(* IEC 61131-3 sources: 2026_Projet_YGO_ExcavatriceDragage/TOOLS/TEST_AUTO_CI/RESULTS/JOYSTICK/tests, 1 file *)

(* ---- test_fb_joystick.st ---- *)
SETUP
VAR
    fb : FB_JOYSTICK;
    nx : INT := 5000;
    ny : INT := 5000;
    diagOk : ST_DIAG_DEVICE;
    diagDown : ST_DIAG_DEVICE;
END_VAR
END_SETUP

TEST 'TC-P08-001 Bus non operationnel neutralise les sorties sans lever Error'
    diagDown.ONLINE := FALSE; diagDown.OPERATIONAL := FALSE; diagDown.ERROR := FALSE;
    diagDown.ERRORID := 0; diagDown.STATE := E_DIAG_STATE.INIT; diagDown.STATEATERROR := E_DIAG_STATE.DISABLED;
    diagOk.ONLINE := TRUE; diagOk.OPERATIONAL := TRUE; diagOk.ERROR := FALSE;
    diagOk.ERRORID := 0; diagOk.STATE := E_DIAG_STATE.READY; diagOk.STATEATERROR := E_DIAG_STATE.DISABLED;

    fb(ENABLE := TRUE, RESET := FALSE, POWERCONTACTORENGAGED := TRUE,
       MODE := E_MODE.MAINT_N1, BENNEBUSY := FALSE, PRESERVEARMINGAFTERBUCKET := FALSE,
       BUSCANOPENOP := diagDown, JOYSTICKOP := diagOk,
       RAWX := 5000, RAWY := 5000, RAWBUTTON := FALSE, BTNCALIBRATE := FALSE,
       INVERTX := FALSE, INVERTY := FALSE, DEADBANDRAW := 300, FILTERTIME := T#0MS,
       NEUTRALHOLDTIME := T#100MS, DEADMANARMHOLDTIME := T#100MS, DEADMANARMGRACETIME := T#3S,
       NEUTRALXMEM := nx, NEUTRALYMEM := ny);

    ASSERT_FALSE(fb.READY, 'bus CAN non operationnel doit bloquer Ready');
    ASSERT_FALSE(fb.ERROR, 'un bus down est un GATE de securite, PAS une Error diagnostiquee (pas de bit ErrorId leve ici)');
    ASSERT_FALSE(fb.AXISCMDX.ENABLE, 'sorties axe neutralisees si non operationnel');
END_TEST

TEST 'TC-P08-002 Appui maintenu 100ms arme le geste (DeadmanArmHoldTime)'
    diagOk.ONLINE := TRUE; diagOk.OPERATIONAL := TRUE; diagOk.ERROR := FALSE;
    diagOk.ERRORID := 0; diagOk.STATE := E_DIAG_STATE.READY; diagOk.STATEATERROR := E_DIAG_STATE.DISABLED;

    (* baseline : neutre, bouton relache *)
    fb(ENABLE := TRUE, RESET := FALSE, POWERCONTACTORENGAGED := TRUE,
       MODE := E_MODE.MAINT_N1, BENNEBUSY := FALSE, PRESERVEARMINGAFTERBUCKET := FALSE,
       BUSCANOPENOP := diagOk, JOYSTICKOP := diagOk,
       RAWX := 5000, RAWY := 5000, RAWBUTTON := FALSE, BTNCALIBRATE := FALSE,
       INVERTX := FALSE, INVERTY := FALSE, DEADBANDRAW := 300, FILTERTIME := T#0MS,
       NEUTRALHOLDTIME := T#100MS, DEADMANARMHOLDTIME := T#100MS, DEADMANARMGRACETIME := T#3S,
       NEUTRALXMEM := nx, NEUTRALYMEM := ny);
    ASSERT_FALSE(fb.DEADMANARMED, 'baseline : bouton relache, pas arme');

    (* front bouton : demarre le maintien, pas encore arme *)
    fb(ENABLE := TRUE, RESET := FALSE, POWERCONTACTORENGAGED := TRUE,
       MODE := E_MODE.MAINT_N1, BENNEBUSY := FALSE, PRESERVEARMINGAFTERBUCKET := FALSE,
       BUSCANOPENOP := diagOk, JOYSTICKOP := diagOk,
       RAWX := 5000, RAWY := 5000, RAWBUTTON := TRUE, BTNCALIBRATE := FALSE,
       INVERTX := FALSE, INVERTY := FALSE, DEADBANDRAW := 300, FILTERTIME := T#0MS,
       NEUTRALHOLDTIME := T#100MS, DEADMANARMHOLDTIME := T#100MS, DEADMANARMGRACETIME := T#3S,
       NEUTRALXMEM := nx, NEUTRALYMEM := ny);
    ASSERT_FALSE(fb.DEADMANARMED, 'front bouton seul ne doit pas armer immediatement (maintien requis)');

    (* 50ms plus tard : maintien pas termine *)
    ADVANCE_TIME(50000000);
    fb(ENABLE := TRUE, RESET := FALSE, POWERCONTACTORENGAGED := TRUE,
       MODE := E_MODE.MAINT_N1, BENNEBUSY := FALSE, PRESERVEARMINGAFTERBUCKET := FALSE,
       BUSCANOPENOP := diagOk, JOYSTICKOP := diagOk,
       RAWX := 5000, RAWY := 5000, RAWBUTTON := TRUE, BTNCALIBRATE := FALSE,
       INVERTX := FALSE, INVERTY := FALSE, DEADBANDRAW := 300, FILTERTIME := T#0MS,
       NEUTRALHOLDTIME := T#100MS, DEADMANARMHOLDTIME := T#100MS, DEADMANARMGRACETIME := T#3S,
       NEUTRALXMEM := nx, NEUTRALYMEM := ny);
    ASSERT_FALSE(fb.DEADMANARMED, '50ms < DeadmanArmHoldTime (100ms) : pas encore arme');

    (* 60ms de plus (total 110ms) : maintien termine -> arme *)
    ADVANCE_TIME(60000000);
    fb(ENABLE := TRUE, RESET := FALSE, POWERCONTACTORENGAGED := TRUE,
       MODE := E_MODE.MAINT_N1, BENNEBUSY := FALSE, PRESERVEARMINGAFTERBUCKET := FALSE,
       BUSCANOPENOP := diagOk, JOYSTICKOP := diagOk,
       RAWX := 5000, RAWY := 5000, RAWBUTTON := TRUE, BTNCALIBRATE := FALSE,
       INVERTX := FALSE, INVERTY := FALSE, DEADBANDRAW := 300, FILTERTIME := T#0MS,
       NEUTRALHOLDTIME := T#100MS, DEADMANARMHOLDTIME := T#100MS, DEADMANARMGRACETIME := T#3S,
       NEUTRALXMEM := nx, NEUTRALYMEM := ny);
    ASSERT_TRUE(fb.DEADMANARMED, '110ms >= DeadmanArmHoldTime (100ms) : geste arme');
END_TEST

TEST 'TC-P08-003 Relachement du bouton avant fin du maintien annule la tentative armement'
    diagOk.ONLINE := TRUE; diagOk.OPERATIONAL := TRUE; diagOk.ERROR := FALSE;
    diagOk.ERRORID := 0; diagOk.STATE := E_DIAG_STATE.READY; diagOk.STATEATERROR := E_DIAG_STATE.DISABLED;

    (* front bouton : demarre le maintien *)
    fb(ENABLE := TRUE, RESET := FALSE, POWERCONTACTORENGAGED := TRUE,
       MODE := E_MODE.MAINT_N1, BENNEBUSY := FALSE, PRESERVEARMINGAFTERBUCKET := FALSE,
       BUSCANOPENOP := diagOk, JOYSTICKOP := diagOk,
       RAWX := 5000, RAWY := 5000, RAWBUTTON := TRUE, BTNCALIBRATE := FALSE,
       INVERTX := FALSE, INVERTY := FALSE, DEADBANDRAW := 300, FILTERTIME := T#0MS,
       NEUTRALHOLDTIME := T#100MS, DEADMANARMHOLDTIME := T#100MS, DEADMANARMGRACETIME := T#3S,
       NEUTRALXMEM := nx, NEUTRALYMEM := ny);

    (* relache a 50ms, avant la fin des 100ms de maintien *)
    ADVANCE_TIME(50000000);
    fb(ENABLE := TRUE, RESET := FALSE, POWERCONTACTORENGAGED := TRUE,
       MODE := E_MODE.MAINT_N1, BENNEBUSY := FALSE, PRESERVEARMINGAFTERBUCKET := FALSE,
       BUSCANOPENOP := diagOk, JOYSTICKOP := diagOk,
       RAWX := 5000, RAWY := 5000, RAWBUTTON := FALSE, BTNCALIBRATE := FALSE,
       INVERTX := FALSE, INVERTY := FALSE, DEADBANDRAW := 300, FILTERTIME := T#0MS,
       NEUTRALHOLDTIME := T#100MS, DEADMANARMHOLDTIME := T#100MS, DEADMANARMGRACETIME := T#3S,
       NEUTRALXMEM := nx, NEUTRALYMEM := ny);
    ASSERT_FALSE(fb.DEADMANARMED, 'relachement avant la fin du maintien annule la tentative');

    (* le bouton reste relache : meme 100ms plus tard, aucun armement differe *)
    ADVANCE_TIME(100000000);
    fb(ENABLE := TRUE, RESET := FALSE, POWERCONTACTORENGAGED := TRUE,
       MODE := E_MODE.MAINT_N1, BENNEBUSY := FALSE, PRESERVEARMINGAFTERBUCKET := FALSE,
       BUSCANOPENOP := diagOk, JOYSTICKOP := diagOk,
       RAWX := 5000, RAWY := 5000, RAWBUTTON := FALSE, BTNCALIBRATE := FALSE,
       INVERTX := FALSE, INVERTY := FALSE, DEADBANDRAW := 300, FILTERTIME := T#0MS,
       NEUTRALHOLDTIME := T#100MS, DEADMANARMHOLDTIME := T#100MS, DEADMANARMGRACETIME := T#3S,
       NEUTRALXMEM := nx, NEUTRALYMEM := ny);
    ASSERT_FALSE(fb.DEADMANARMED, 'pas d armement differe sur une tentative deja annulee (nouvel appui conscient exige)');

    (* nouveau front + maintien complet : l armement redevient possible normalement *)
    ADVANCE_TIME(10000000);
    fb(ENABLE := TRUE, RESET := FALSE, POWERCONTACTORENGAGED := TRUE,
       MODE := E_MODE.MAINT_N1, BENNEBUSY := FALSE, PRESERVEARMINGAFTERBUCKET := FALSE,
       BUSCANOPENOP := diagOk, JOYSTICKOP := diagOk,
       RAWX := 5000, RAWY := 5000, RAWBUTTON := TRUE, BTNCALIBRATE := FALSE,
       INVERTX := FALSE, INVERTY := FALSE, DEADBANDRAW := 300, FILTERTIME := T#0MS,
       NEUTRALHOLDTIME := T#100MS, DEADMANARMHOLDTIME := T#100MS, DEADMANARMGRACETIME := T#3S,
       NEUTRALXMEM := nx, NEUTRALYMEM := ny);
    ADVANCE_TIME(110000000);
    fb(ENABLE := TRUE, RESET := FALSE, POWERCONTACTORENGAGED := TRUE,
       MODE := E_MODE.MAINT_N1, BENNEBUSY := FALSE, PRESERVEARMINGAFTERBUCKET := FALSE,
       BUSCANOPENOP := diagOk, JOYSTICKOP := diagOk,
       RAWX := 5000, RAWY := 5000, RAWBUTTON := TRUE, BTNCALIBRATE := FALSE,
       INVERTX := FALSE, INVERTY := FALSE, DEADBANDRAW := 300, FILTERTIME := T#0MS,
       NEUTRALHOLDTIME := T#100MS, DEADMANARMHOLDTIME := T#100MS, DEADMANARMGRACETIME := T#3S,
       NEUTRALXMEM := nx, NEUTRALYMEM := ny);
    ASSERT_TRUE(fb.DEADMANARMED, 'un nouvel appui complet doit toujours pouvoir armer');
END_TEST

TEST 'TC-P08-004 Delai de grace protege l armement au neutre, puis le neutre prolonge desarme apres la grace'
    diagOk.ONLINE := TRUE; diagOk.OPERATIONAL := TRUE; diagOk.ERROR := FALSE;
    diagOk.ERRORID := 0; diagOk.STATE := E_DIAG_STATE.READY; diagOk.STATEATERROR := E_DIAG_STATE.DISABLED;

    (* nx/ny fixes explicitement a 5000 avant CHAQUE appel : STruCpp ne re-copie PAS la sortie
       VAR_IN_OUT vers la variable de test entre deux appels fb() (limite outillage constatee,
       round-trip IN_OUT absent -- cf. README). Sans ce forcage, NeutralXMem retomberait a 0
       (valeur SETUP jamais appliquee non plus) des le 2e scan, et AtNeutral resterait FALSE. *)
    nx := 5000; ny := 5000;

    (* arme le geste au neutre *)
    fb(ENABLE := TRUE, RESET := FALSE, POWERCONTACTORENGAGED := TRUE,
       MODE := E_MODE.MAINT_N1, BENNEBUSY := FALSE, PRESERVEARMINGAFTERBUCKET := FALSE,
       BUSCANOPENOP := diagOk, JOYSTICKOP := diagOk,
       RAWX := 5000, RAWY := 5000, RAWBUTTON := TRUE, BTNCALIBRATE := FALSE,
       INVERTX := FALSE, INVERTY := FALSE, DEADBANDRAW := 300, FILTERTIME := T#0MS,
       NEUTRALHOLDTIME := T#100MS, DEADMANARMHOLDTIME := T#100MS, DEADMANARMGRACETIME := T#3S,
       NEUTRALXMEM := nx, NEUTRALYMEM := ny);
    ADVANCE_TIME(110000000);
    fb(ENABLE := TRUE, RESET := FALSE, POWERCONTACTORENGAGED := TRUE,
       MODE := E_MODE.MAINT_N1, BENNEBUSY := FALSE, PRESERVEARMINGAFTERBUCKET := FALSE,
       BUSCANOPENOP := diagOk, JOYSTICKOP := diagOk,
       RAWX := 5000, RAWY := 5000, RAWBUTTON := TRUE, BTNCALIBRATE := FALSE,
       INVERTX := FALSE, INVERTY := FALSE, DEADBANDRAW := 300, FILTERTIME := T#0MS,
       NEUTRALHOLDTIME := T#100MS, DEADMANARMHOLDTIME := T#100MS, DEADMANARMGRACETIME := T#3S,
       NEUTRALXMEM := nx, NEUTRALYMEM := ny);
    ASSERT_TRUE(fb.DEADMANARMED, 'precondition : geste arme');

    (* bouton relache, reste au neutre : 500ms plus tard (largement > NeutralHoldTime seul 100ms) mais < grace (3s) *)
    ADVANCE_TIME(500000000);
    fb(ENABLE := TRUE, RESET := FALSE, POWERCONTACTORENGAGED := TRUE,
       MODE := E_MODE.MAINT_N1, BENNEBUSY := FALSE, PRESERVEARMINGAFTERBUCKET := FALSE,
       BUSCANOPENOP := diagOk, JOYSTICKOP := diagOk,
       RAWX := 5000, RAWY := 5000, RAWBUTTON := FALSE, BTNCALIBRATE := FALSE,
       INVERTX := FALSE, INVERTY := FALSE, DEADBANDRAW := 300, FILTERTIME := T#0MS,
       NEUTRALHOLDTIME := T#100MS, DEADMANARMHOLDTIME := T#100MS, DEADMANARMGRACETIME := T#3S,
       NEUTRALXMEM := nx, NEUTRALYMEM := ny);
    ASSERT_TRUE(fb.DEADMANARMED, 'la grace (3s) protege l armement malgre un neutre deja tenu bien plus longtemps que NeutralHoldTime seul (evite le REX terrain : desarmement 100-200ms apres l armement)');

    (* 2.6s de plus (total 3.1s depuis l armement) : la grace vient de s ecouler ce scan meme --
       NeutralHoldTimer ne fait que DEMARRER (son IN passe a TRUE ce scan), pas encore Q *)
    ADVANCE_TIME(2600000000);
    fb(ENABLE := TRUE, RESET := FALSE, POWERCONTACTORENGAGED := TRUE,
       MODE := E_MODE.MAINT_N1, BENNEBUSY := FALSE, PRESERVEARMINGAFTERBUCKET := FALSE,
       BUSCANOPENOP := diagOk, JOYSTICKOP := diagOk,
       RAWX := 5000, RAWY := 5000, RAWBUTTON := FALSE, BTNCALIBRATE := FALSE,
       INVERTX := FALSE, INVERTY := FALSE, DEADBANDRAW := 300, FILTERTIME := T#0MS,
       NEUTRALHOLDTIME := T#100MS, DEADMANARMHOLDTIME := T#100MS, DEADMANARMGRACETIME := T#3S,
       NEUTRALXMEM := nx, NEUTRALYMEM := ny);
    ASSERT_TRUE(fb.DEADMANARMED, 'grace tout juste ecoulee : NeutralHoldTimer demarre seulement ce scan (pas encore ecoule)');

    (* 100ms de plus (NeutralHoldTime ecoule depuis la fin de la grace) : desarme *)
    ADVANCE_TIME(100000000);
    fb(ENABLE := TRUE, RESET := FALSE, POWERCONTACTORENGAGED := TRUE,
       MODE := E_MODE.MAINT_N1, BENNEBUSY := FALSE, PRESERVEARMINGAFTERBUCKET := FALSE,
       BUSCANOPENOP := diagOk, JOYSTICKOP := diagOk,
       RAWX := 5000, RAWY := 5000, RAWBUTTON := FALSE, BTNCALIBRATE := FALSE,
       INVERTX := FALSE, INVERTY := FALSE, DEADBANDRAW := 300, FILTERTIME := T#0MS,
       NEUTRALHOLDTIME := T#100MS, DEADMANARMHOLDTIME := T#100MS, DEADMANARMGRACETIME := T#3S,
       NEUTRALXMEM := nx, NEUTRALYMEM := ny);
    ASSERT_FALSE(fb.DEADMANARMED, 'grace ecoulee (3s) + neutre tenu (NeutralHoldTime) : desarmement');
END_TEST

TEST 'TC-P08-005 Changement de mode desarme le geste, nouvel appui exige'
    diagOk.ONLINE := TRUE; diagOk.OPERATIONAL := TRUE; diagOk.ERROR := FALSE;
    diagOk.ERRORID := 0; diagOk.STATE := E_DIAG_STATE.READY; diagOk.STATEATERROR := E_DIAG_STATE.DISABLED;

    (* arme en MAINT_N1 *)
    fb(ENABLE := TRUE, RESET := FALSE, POWERCONTACTORENGAGED := TRUE,
       MODE := E_MODE.MAINT_N1, BENNEBUSY := FALSE, PRESERVEARMINGAFTERBUCKET := FALSE,
       BUSCANOPENOP := diagOk, JOYSTICKOP := diagOk,
       RAWX := 5000, RAWY := 5000, RAWBUTTON := TRUE, BTNCALIBRATE := FALSE,
       INVERTX := FALSE, INVERTY := FALSE, DEADBANDRAW := 300, FILTERTIME := T#0MS,
       NEUTRALHOLDTIME := T#100MS, DEADMANARMHOLDTIME := T#100MS, DEADMANARMGRACETIME := T#3S,
       NEUTRALXMEM := nx, NEUTRALYMEM := ny);
    ADVANCE_TIME(110000000);
    fb(ENABLE := TRUE, RESET := FALSE, POWERCONTACTORENGAGED := TRUE,
       MODE := E_MODE.MAINT_N1, BENNEBUSY := FALSE, PRESERVEARMINGAFTERBUCKET := FALSE,
       BUSCANOPENOP := diagOk, JOYSTICKOP := diagOk,
       RAWX := 5000, RAWY := 5000, RAWBUTTON := TRUE, BTNCALIBRATE := FALSE,
       INVERTX := FALSE, INVERTY := FALSE, DEADBANDRAW := 300, FILTERTIME := T#0MS,
       NEUTRALHOLDTIME := T#100MS, DEADMANARMHOLDTIME := T#100MS, DEADMANARMGRACETIME := T#3S,
       NEUTRALXMEM := nx, NEUTRALYMEM := ny);
    ASSERT_TRUE(fb.DEADMANARMED, 'precondition : geste arme');

    (* changement de mode : desarmement immediat *)
    ADVANCE_TIME(10000000);
    fb(ENABLE := TRUE, RESET := FALSE, POWERCONTACTORENGAGED := TRUE,
       MODE := E_MODE.MAINT_N2, BENNEBUSY := FALSE, PRESERVEARMINGAFTERBUCKET := FALSE,
       BUSCANOPENOP := diagOk, JOYSTICKOP := diagOk,
       RAWX := 5000, RAWY := 5000, RAWBUTTON := FALSE, BTNCALIBRATE := FALSE,
       INVERTX := FALSE, INVERTY := FALSE, DEADBANDRAW := 300, FILTERTIME := T#0MS,
       NEUTRALHOLDTIME := T#100MS, DEADMANARMHOLDTIME := T#100MS, DEADMANARMGRACETIME := T#3S,
       NEUTRALXMEM := nx, NEUTRALYMEM := ny);
    ASSERT_FALSE(fb.DEADMANARMED, 'changement de mode desarme immediatement');

    (* mode stable ensuite, sans nouvel appui : reste desarme *)
    ADVANCE_TIME(10000000);
    fb(ENABLE := TRUE, RESET := FALSE, POWERCONTACTORENGAGED := TRUE,
       MODE := E_MODE.MAINT_N2, BENNEBUSY := FALSE, PRESERVEARMINGAFTERBUCKET := FALSE,
       BUSCANOPENOP := diagOk, JOYSTICKOP := diagOk,
       RAWX := 5000, RAWY := 5000, RAWBUTTON := FALSE, BTNCALIBRATE := FALSE,
       INVERTX := FALSE, INVERTY := FALSE, DEADBANDRAW := 300, FILTERTIME := T#0MS,
       NEUTRALHOLDTIME := T#100MS, DEADMANARMHOLDTIME := T#100MS, DEADMANARMGRACETIME := T#3S,
       NEUTRALXMEM := nx, NEUTRALYMEM := ny);
    ASSERT_FALSE(fb.DEADMANARMED, 'pas de rearmement automatique apres changement de mode : nouvel appui conscient exige');
END_TEST

TEST 'TC-P08-006 Reset acquitte une erreur de calibration seulement si la cause a disparu'
    diagOk.ONLINE := TRUE; diagOk.OPERATIONAL := TRUE; diagOk.ERROR := FALSE;
    diagOk.ERRORID := 0; diagOk.STATE := E_DIAG_STATE.READY; diagOk.STATEATERROR := E_DIAG_STATE.DISABLED;

    (* RawX/RawY hors zone neutre valide (2000..8000) + front BtnCalibrate *)
    fb(ENABLE := TRUE, RESET := FALSE, POWERCONTACTORENGAGED := TRUE,
       MODE := E_MODE.MAINT_N1, BENNEBUSY := FALSE, PRESERVEARMINGAFTERBUCKET := FALSE,
       BUSCANOPENOP := diagOk, JOYSTICKOP := diagOk,
       RAWX := 9500, RAWY := 9500, RAWBUTTON := FALSE, BTNCALIBRATE := FALSE,
       INVERTX := FALSE, INVERTY := FALSE, DEADBANDRAW := 300, FILTERTIME := T#0MS,
       NEUTRALHOLDTIME := T#100MS, DEADMANARMHOLDTIME := T#100MS, DEADMANARMGRACETIME := T#3S,
       NEUTRALXMEM := nx, NEUTRALYMEM := ny);

    fb(ENABLE := TRUE, RESET := FALSE, POWERCONTACTORENGAGED := TRUE,
       MODE := E_MODE.MAINT_N1, BENNEBUSY := FALSE, PRESERVEARMINGAFTERBUCKET := FALSE,
       BUSCANOPENOP := diagOk, JOYSTICKOP := diagOk,
       RAWX := 9500, RAWY := 9500, RAWBUTTON := FALSE, BTNCALIBRATE := TRUE,
       INVERTX := FALSE, INVERTY := FALSE, DEADBANDRAW := 300, FILTERTIME := T#0MS,
       NEUTRALHOLDTIME := T#100MS, DEADMANARMHOLDTIME := T#100MS, DEADMANARMGRACETIME := T#3S,
       NEUTRALXMEM := nx, NEUTRALYMEM := ny);

    ASSERT_TRUE(fb.ERROR, 'calibration hors zone doit lever Error');

    (* Reset alors que la cause est toujours presente (axes toujours hors zone) : ne doit PAS acquitter *)
    fb(ENABLE := TRUE, RESET := TRUE, POWERCONTACTORENGAGED := TRUE,
       MODE := E_MODE.MAINT_N1, BENNEBUSY := FALSE, PRESERVEARMINGAFTERBUCKET := FALSE,
       BUSCANOPENOP := diagOk, JOYSTICKOP := diagOk,
       RAWX := 9500, RAWY := 9500, RAWBUTTON := FALSE, BTNCALIBRATE := FALSE,
       INVERTX := FALSE, INVERTY := FALSE, DEADBANDRAW := 300, FILTERTIME := T#0MS,
       NEUTRALHOLDTIME := T#100MS, DEADMANARMHOLDTIME := T#100MS, DEADMANARMGRACETIME := T#3S,
       NEUTRALXMEM := nx, NEUTRALYMEM := ny);

    ASSERT_TRUE(fb.ERROR, 'Reset ne doit PAS acquitter tant que les axes restent hors zone (cause toujours presente)');

    (* Reset retombe (front consomme) ; axes reviennent en zone ; nouveau front Reset : doit acquitter *)
    fb(ENABLE := TRUE, RESET := FALSE, POWERCONTACTORENGAGED := TRUE,
       MODE := E_MODE.MAINT_N1, BENNEBUSY := FALSE, PRESERVEARMINGAFTERBUCKET := FALSE,
       BUSCANOPENOP := diagOk, JOYSTICKOP := diagOk,
       RAWX := 5000, RAWY := 5000, RAWBUTTON := FALSE, BTNCALIBRATE := FALSE,
       INVERTX := FALSE, INVERTY := FALSE, DEADBANDRAW := 300, FILTERTIME := T#0MS,
       NEUTRALHOLDTIME := T#100MS, DEADMANARMHOLDTIME := T#100MS, DEADMANARMGRACETIME := T#3S,
       NEUTRALXMEM := nx, NEUTRALYMEM := ny);

    fb(ENABLE := TRUE, RESET := TRUE, POWERCONTACTORENGAGED := TRUE,
       MODE := E_MODE.MAINT_N1, BENNEBUSY := FALSE, PRESERVEARMINGAFTERBUCKET := FALSE,
       BUSCANOPENOP := diagOk, JOYSTICKOP := diagOk,
       RAWX := 5000, RAWY := 5000, RAWBUTTON := FALSE, BTNCALIBRATE := FALSE,
       INVERTX := FALSE, INVERTY := FALSE, DEADBANDRAW := 300, FILTERTIME := T#0MS,
       NEUTRALHOLDTIME := T#100MS, DEADMANARMHOLDTIME := T#100MS, DEADMANARMGRACETIME := T#3S,
       NEUTRALXMEM := nx, NEUTRALYMEM := ny);

    ASSERT_FALSE(fb.ERROR, 'front Reset avec axes revenus en zone valide doit acquitter (cause disparue + appui conscient)');
END_TEST

TEST 'TC-P08-007 SpeedRef sature a +/-100 meme avec RawX/RawY hors plage nominale (defaut capteur)'
    diagOk.ONLINE := TRUE; diagOk.OPERATIONAL := TRUE; diagOk.ERROR := FALSE;
    diagOk.ERRORID := 0; diagOk.STATE := E_DIAG_STATE.READY; diagOk.STATEATERROR := E_DIAG_STATE.DISABLED;
    (* init explicite -- STruCpp n applique pas ":= 5000" du SETUP, cf. README limite outillage *)
    nx := 5000; ny := 5000;

    (* arme le geste au neutre *)
    fb(ENABLE := TRUE, RESET := FALSE, POWERCONTACTORENGAGED := TRUE,
       MODE := E_MODE.MAINT_N1, BENNEBUSY := FALSE, PRESERVEARMINGAFTERBUCKET := FALSE,
       BUSCANOPENOP := diagOk, JOYSTICKOP := diagOk,
       RAWX := 5000, RAWY := 5000, RAWBUTTON := TRUE, BTNCALIBRATE := FALSE,
       INVERTX := FALSE, INVERTY := FALSE, DEADBANDRAW := 300, FILTERTIME := T#0MS,
       NEUTRALHOLDTIME := T#100MS, DEADMANARMHOLDTIME := T#100MS, DEADMANARMGRACETIME := T#3S,
       NEUTRALXMEM := nx, NEUTRALYMEM := ny);
    ADVANCE_TIME(110000000);
    fb(ENABLE := TRUE, RESET := FALSE, POWERCONTACTORENGAGED := TRUE,
       MODE := E_MODE.MAINT_N1, BENNEBUSY := FALSE, PRESERVEARMINGAFTERBUCKET := FALSE,
       BUSCANOPENOP := diagOk, JOYSTICKOP := diagOk,
       RAWX := 5000, RAWY := 5000, RAWBUTTON := TRUE, BTNCALIBRATE := FALSE,
       INVERTX := FALSE, INVERTY := FALSE, DEADBANDRAW := 300, FILTERTIME := T#0MS,
       NEUTRALHOLDTIME := T#100MS, DEADMANARMHOLDTIME := T#100MS, DEADMANARMGRACETIME := T#3S,
       NEUTRALXMEM := nx, NEUTRALYMEM := ny);
    ASSERT_TRUE(fb.DEADMANARMED, 'precondition : geste arme');

    (* RawX/RawY au maximum nominal (10000) : saturation +100 *)
    ADVANCE_TIME(10000000);
    fb(ENABLE := TRUE, RESET := FALSE, POWERCONTACTORENGAGED := TRUE,
       MODE := E_MODE.MAINT_N1, BENNEBUSY := FALSE, PRESERVEARMINGAFTERBUCKET := FALSE,
       BUSCANOPENOP := diagOk, JOYSTICKOP := diagOk,
       RAWX := 10000, RAWY := 10000, RAWBUTTON := FALSE, BTNCALIBRATE := FALSE,
       INVERTX := FALSE, INVERTY := FALSE, DEADBANDRAW := 300, FILTERTIME := T#0MS,
       NEUTRALHOLDTIME := T#100MS, DEADMANARMHOLDTIME := T#100MS, DEADMANARMGRACETIME := T#3S,
       NEUTRALXMEM := nx, NEUTRALYMEM := ny);
    ASSERT_NEAR(fb.AXISCMDX.SPEEDREF, 100.0, 0.01, 'RawX au max nominal (10000) : SpeedRef sature a +100');
    ASSERT_NEAR(fb.AXISCMDY.SPEEDREF, 100.0, 0.01, 'meme comportement sur l axe Y');
    ASSERT_EQ(fb.AXISCMDX.DIRECTION, 1, 'Direction coherente avec le signe de la consigne');

    (* RawX/RawY au minimum nominal (0) : saturation -100 *)
    ADVANCE_TIME(10000000);
    fb(ENABLE := TRUE, RESET := FALSE, POWERCONTACTORENGAGED := TRUE,
       MODE := E_MODE.MAINT_N1, BENNEBUSY := FALSE, PRESERVEARMINGAFTERBUCKET := FALSE,
       BUSCANOPENOP := diagOk, JOYSTICKOP := diagOk,
       RAWX := 0, RAWY := 0, RAWBUTTON := FALSE, BTNCALIBRATE := FALSE,
       INVERTX := FALSE, INVERTY := FALSE, DEADBANDRAW := 300, FILTERTIME := T#0MS,
       NEUTRALHOLDTIME := T#100MS, DEADMANARMHOLDTIME := T#100MS, DEADMANARMGRACETIME := T#3S,
       NEUTRALXMEM := nx, NEUTRALYMEM := ny);
    ASSERT_NEAR(fb.AXISCMDX.SPEEDREF, -100.0, 0.01, 'RawX au min nominal (0) : SpeedRef sature a -100');
    ASSERT_EQ(fb.AXISCMDX.DIRECTION, -1, 'Direction coherente avec le signe de la consigne');

    (* Depassement franc au-dela de la plage ADC nominale (defaut capteur/cablage Hall) :
       le garde-fou LIMIT(-100,OutPct,100) de FB_AxisScale doit clamper, jamais deborder *)
    ADVANCE_TIME(10000000);
    fb(ENABLE := TRUE, RESET := FALSE, POWERCONTACTORENGAGED := TRUE,
       MODE := E_MODE.MAINT_N1, BENNEBUSY := FALSE, PRESERVEARMINGAFTERBUCKET := FALSE,
       BUSCANOPENOP := diagOk, JOYSTICKOP := diagOk,
       RAWX := 20000, RAWY := 20000, RAWBUTTON := FALSE, BTNCALIBRATE := FALSE,
       INVERTX := FALSE, INVERTY := FALSE, DEADBANDRAW := 300, FILTERTIME := T#0MS,
       NEUTRALHOLDTIME := T#100MS, DEADMANARMHOLDTIME := T#100MS, DEADMANARMGRACETIME := T#3S,
       NEUTRALXMEM := nx, NEUTRALYMEM := ny);
    ASSERT_NEAR(fb.AXISCMDX.SPEEDREF, 100.0, 0.01, 'RawX=20000 (hors plage ADC 0..10000, defaut capteur) : toujours clampe a +100, pas de debordement');
    ASSERT_NEAR(fb.AXISCMDY.SPEEDREF, 100.0, 0.01, 'meme garde-fou sur l axe Y');

    (* Valeur negative (hors plage ADC, meme scenario defaut cablage) *)
    ADVANCE_TIME(10000000);
    fb(ENABLE := TRUE, RESET := FALSE, POWERCONTACTORENGAGED := TRUE,
       MODE := E_MODE.MAINT_N1, BENNEBUSY := FALSE, PRESERVEARMINGAFTERBUCKET := FALSE,
       BUSCANOPENOP := diagOk, JOYSTICKOP := diagOk,
       RAWX := -10000, RAWY := -10000, RAWBUTTON := FALSE, BTNCALIBRATE := FALSE,
       INVERTX := FALSE, INVERTY := FALSE, DEADBANDRAW := 300, FILTERTIME := T#0MS,
       NEUTRALHOLDTIME := T#100MS, DEADMANARMHOLDTIME := T#100MS, DEADMANARMGRACETIME := T#3S,
       NEUTRALXMEM := nx, NEUTRALYMEM := ny);
    ASSERT_NEAR(fb.AXISCMDX.SPEEDREF, -100.0, 0.01, 'RawX negatif (hors plage ADC, defaut capteur) : toujours clampe a -100, pas de debordement');
    ASSERT_NEAR(fb.AXISCMDY.SPEEDREF, -100.0, 0.01, 'meme garde-fou sur l axe Y');
END_TEST

TEST 'TC-P08-011 Fin de cycle benne desarme le geste par defaut'
    diagOk.ONLINE := TRUE; diagOk.OPERATIONAL := TRUE; diagOk.ERROR := FALSE;
    diagOk.ERRORID := 0; diagOk.STATE := E_DIAG_STATE.READY; diagOk.STATEATERROR := E_DIAG_STATE.DISABLED;

    (* arme le geste *)
    fb(ENABLE := TRUE, RESET := FALSE, POWERCONTACTORENGAGED := TRUE,
       MODE := E_MODE.MAINT_N1, BENNEBUSY := FALSE, PRESERVEARMINGAFTERBUCKET := FALSE,
       BUSCANOPENOP := diagOk, JOYSTICKOP := diagOk,
       RAWX := 5000, RAWY := 5000, RAWBUTTON := TRUE, BTNCALIBRATE := FALSE,
       INVERTX := FALSE, INVERTY := FALSE, DEADBANDRAW := 300, FILTERTIME := T#0MS,
       NEUTRALHOLDTIME := T#100MS, DEADMANARMHOLDTIME := T#100MS, DEADMANARMGRACETIME := T#3S,
       NEUTRALXMEM := nx, NEUTRALYMEM := ny);
    ADVANCE_TIME(110000000);
    fb(ENABLE := TRUE, RESET := FALSE, POWERCONTACTORENGAGED := TRUE,
       MODE := E_MODE.MAINT_N1, BENNEBUSY := FALSE, PRESERVEARMINGAFTERBUCKET := FALSE,
       BUSCANOPENOP := diagOk, JOYSTICKOP := diagOk,
       RAWX := 5000, RAWY := 5000, RAWBUTTON := TRUE, BTNCALIBRATE := FALSE,
       INVERTX := FALSE, INVERTY := FALSE, DEADBANDRAW := 300, FILTERTIME := T#0MS,
       NEUTRALHOLDTIME := T#100MS, DEADMANARMHOLDTIME := T#100MS, DEADMANARMGRACETIME := T#3S,
       NEUTRALXMEM := nx, NEUTRALYMEM := ny);
    ASSERT_TRUE(fb.DEADMANARMED, 'precondition : geste arme');

    (* BenneBusy actif : ne desarme pas seul (attend le front descendant) *)
    ADVANCE_TIME(10000000);
    fb(ENABLE := TRUE, RESET := FALSE, POWERCONTACTORENGAGED := TRUE,
       MODE := E_MODE.MAINT_N1, BENNEBUSY := TRUE, PRESERVEARMINGAFTERBUCKET := FALSE,
       BUSCANOPENOP := diagOk, JOYSTICKOP := diagOk,
       RAWX := 5000, RAWY := 5000, RAWBUTTON := FALSE, BTNCALIBRATE := FALSE,
       INVERTX := FALSE, INVERTY := FALSE, DEADBANDRAW := 300, FILTERTIME := T#0MS,
       NEUTRALHOLDTIME := T#100MS, DEADMANARMHOLDTIME := T#100MS, DEADMANARMGRACETIME := T#3S,
       NEUTRALXMEM := nx, NEUTRALYMEM := ny);
    ASSERT_TRUE(fb.DEADMANARMED, 'BenneBusy actif seul ne desarme pas (attend le front descendant, fin de cycle)');

    (* front descendant BenneBusy, sans exception : desarme immediatement *)
    ADVANCE_TIME(10000000);
    fb(ENABLE := TRUE, RESET := FALSE, POWERCONTACTORENGAGED := TRUE,
       MODE := E_MODE.MAINT_N1, BENNEBUSY := FALSE, PRESERVEARMINGAFTERBUCKET := FALSE,
       BUSCANOPENOP := diagOk, JOYSTICKOP := diagOk,
       RAWX := 5000, RAWY := 5000, RAWBUTTON := FALSE, BTNCALIBRATE := FALSE,
       INVERTX := FALSE, INVERTY := FALSE, DEADBANDRAW := 300, FILTERTIME := T#0MS,
       NEUTRALHOLDTIME := T#100MS, DEADMANARMHOLDTIME := T#100MS, DEADMANARMGRACETIME := T#3S,
       NEUTRALXMEM := nx, NEUTRALYMEM := ny);
    ASSERT_FALSE(fb.DEADMANARMED, 'front descendant BenneBusy sans exception desarme immediatement (pas de M1/M2 surprise)');
END_TEST

TEST 'TC-P08-012 PreserveArmingAfterBucket protege l armement en fin de benne (exception CLOSING Extraction)'
    diagOk.ONLINE := TRUE; diagOk.OPERATIONAL := TRUE; diagOk.ERROR := FALSE;
    diagOk.ERRORID := 0; diagOk.STATE := E_DIAG_STATE.READY; diagOk.STATEATERROR := E_DIAG_STATE.DISABLED;

    (* arme le geste *)
    fb(ENABLE := TRUE, RESET := FALSE, POWERCONTACTORENGAGED := TRUE,
       MODE := E_MODE.MAINT_N1, BENNEBUSY := FALSE, PRESERVEARMINGAFTERBUCKET := FALSE,
       BUSCANOPENOP := diagOk, JOYSTICKOP := diagOk,
       RAWX := 5000, RAWY := 5000, RAWBUTTON := TRUE, BTNCALIBRATE := FALSE,
       INVERTX := FALSE, INVERTY := FALSE, DEADBANDRAW := 300, FILTERTIME := T#0MS,
       NEUTRALHOLDTIME := T#100MS, DEADMANARMHOLDTIME := T#100MS, DEADMANARMGRACETIME := T#3S,
       NEUTRALXMEM := nx, NEUTRALYMEM := ny);
    ADVANCE_TIME(110000000);
    fb(ENABLE := TRUE, RESET := FALSE, POWERCONTACTORENGAGED := TRUE,
       MODE := E_MODE.MAINT_N1, BENNEBUSY := FALSE, PRESERVEARMINGAFTERBUCKET := FALSE,
       BUSCANOPENOP := diagOk, JOYSTICKOP := diagOk,
       RAWX := 5000, RAWY := 5000, RAWBUTTON := TRUE, BTNCALIBRATE := FALSE,
       INVERTX := FALSE, INVERTY := FALSE, DEADBANDRAW := 300, FILTERTIME := T#0MS,
       NEUTRALHOLDTIME := T#100MS, DEADMANARMHOLDTIME := T#100MS, DEADMANARMGRACETIME := T#3S,
       NEUTRALXMEM := nx, NEUTRALYMEM := ny);
    ASSERT_TRUE(fb.DEADMANARMED, 'precondition : geste arme');

    (* BenneBusy actif, exception active *)
    ADVANCE_TIME(10000000);
    fb(ENABLE := TRUE, RESET := FALSE, POWERCONTACTORENGAGED := TRUE,
       MODE := E_MODE.MAINT_N1, BENNEBUSY := TRUE, PRESERVEARMINGAFTERBUCKET := TRUE,
       BUSCANOPENOP := diagOk, JOYSTICKOP := diagOk,
       RAWX := 5000, RAWY := 5000, RAWBUTTON := FALSE, BTNCALIBRATE := FALSE,
       INVERTX := FALSE, INVERTY := FALSE, DEADBANDRAW := 300, FILTERTIME := T#0MS,
       NEUTRALHOLDTIME := T#100MS, DEADMANARMHOLDTIME := T#100MS, DEADMANARMGRACETIME := T#3S,
       NEUTRALXMEM := nx, NEUTRALYMEM := ny);

    (* front descendant BenneBusy, exception active : l armement doit etre conserve *)
    ADVANCE_TIME(10000000);
    fb(ENABLE := TRUE, RESET := FALSE, POWERCONTACTORENGAGED := TRUE,
       MODE := E_MODE.MAINT_N1, BENNEBUSY := FALSE, PRESERVEARMINGAFTERBUCKET := TRUE,
       BUSCANOPENOP := diagOk, JOYSTICKOP := diagOk,
       RAWX := 5000, RAWY := 5000, RAWBUTTON := FALSE, BTNCALIBRATE := FALSE,
       INVERTX := FALSE, INVERTY := FALSE, DEADBANDRAW := 300, FILTERTIME := T#0MS,
       NEUTRALHOLDTIME := T#100MS, DEADMANARMHOLDTIME := T#100MS, DEADMANARMGRACETIME := T#3S,
       NEUTRALXMEM := nx, NEUTRALYMEM := ny);
    ASSERT_TRUE(fb.DEADMANARMED, 'PreserveArmingAfterBucket=TRUE : armement conserve malgre la fin de benne (exception documentee AF, alerte P1 : ne jamais elargir hors CLOSING Extraction)');
END_TEST
